TYPE T_Ctrl_SIf_MOD_Cur :
STRUCT
	///[ms] time last cycle
	udiCycleTime_ms: UDINT;
END_STRUCT
END_TYPE

(* stored: Version 1.1.0.1, ProductVersion 3.1.0.14
   DUT T_Ctrl_SIf_MOD_Cur: Id {2265d463-493c-42d1-9ba6-86c7d9b8a41f} *)
